TYPE FaulhaberDriveStatuses :
STRUCT
	///Is the NcAxis in a busy state?
	busyStatus: BusyStatus;
	///Is the NcAxis in a healthy state?
	healthStatus: HealthStatus;
END_STRUCT
END_TYPE

(* stored: Version 1.1.0.1, ProductVersion 3.1.4019.2
   DUT FaulhaberDriveStatuses: Id {4fd3450c-339c-43e9-9d3f-53745a5b5006} *)
